(* IEC 61131-3 sources: Elmo_Master/Lasal_PRG/MotionTCPDemo/Class/TCPRT_DataManager, 1 file *)

(* ---- TCPRT_DataManager.st ---- *)
(*!
<Class
	Name               = "TCPRT_DataManager"
	Revision           = "0.0"
	RealtimeTask       = "true"
	CyclicTask         = "true"
	BackgroundTask     = "false"
	Sigmatek           = "false"
	OSInterface        = "false"
	HighPriority       = "false"
	Automatic          = "false"
	UpdateMode         = "Prescan"
	SharedCommandTable = "true"
	Objectsize         = "(678,0)">
	<Channels>
	</Channels>
	<Network Name="TCPRT_DataManager">
		<!-- List of Components in this network -->
		<Components>
			<Object
				Name       = "_base"
				Class      = "_SigTCPDataManager"
				Position   = "(218,120)"
				Visualized = "true"
				Remotely   = "true">
				<Channels>
					<Server Name="AcceptOfflineJobs" Value="1"/>
					<Server Name="ClassSvr"/>
					<Server Name="ComPort" Value="500"/>
					<Server Name="DeactivateCom" Value="0"/>
					<Server Name="DeleteJobs"/>
					<Server Name="LogEnable" Value="0"/>
					<Server Name="NoEntries"/>
					<Server Name="Online"/>
					<Server Name="ResetLogBuffer"/>
					<Server Name="TCPComm"/>
					<Client Name="ErrRuntime"/>
					<Client Name="InternConnection"/>
					<Client Name="IPtoConnect"/>
					<Client Name="LogFilter" Value="0"/>
					<Client Name="SizeOfComBufferRecv" Value="100 kB"/>
					<Client Name="SizeOfComBuffers" Value="100 kB"/>
					<Client Name="StationToConnect"/>
				</Channels>
			</Object>
		</Components>
		<Comments>
		</Comments>
		<!-- List of Connections in this network -->
		<Connections>
			<Connection Source="this.ClassSvr" Destination="_base.ClassSvr" Vertices="(1084,210),(912,210),"/>
			<Connection Source="this.NoEntries" Destination="_base.NoEntries" Vertices="(1084,270),(912,270),"/>
			<Connection Source="this.DeleteJobs" Destination="_base.DeleteJobs" Vertices="(1084,330),(912,330),"/>
			<Connection Source="this.AcceptOfflineJobs" Destination="_base.AcceptOfflineJobs" Vertices="(1084,390),(912,390),"/>
			<Connection Source="this.TCPComm" Destination="_base.TCPComm" Vertices="(1084,450),(912,510),"/>
			<Connection Source="this.ComPort" Destination="_base.ComPort" Vertices="(1084,510),(912,570),"/>
			<Connection Source="this.Online" Destination="_base.Online" Vertices="(1084,570),(912,630),"/>
			<Connection Source="this.LogEnable" Destination="_base.LogEnable" Vertices="(1084,630),(912,690),"/>
			<Connection Source="this.ResetLogBuffer" Destination="_base.ResetLogBuffer" Vertices="(1084,690),(912,750),"/>
			<Connection Source="this.DeactivateCom" Destination="_base.DeactivateCom" Vertices="(1084,750),(912,810),"/>
			<Connection Source="_base.InternConnection" Destination="this.InternConnection" Vertices="(218,210),(38,210),"/>
			<Connection Source="_base.IPtoConnect" Destination="this.IPtoConnect" Vertices="(218,270),(38,270),"/>
			<Connection Source="_base.StationToConnect" Destination="this.StationToConnect" Vertices="(218,330),(38,330),"/>
			<Connection Source="_base.LogFilter" Destination="this.LogFilter" Vertices="(218,390),(38,390),"/>
			<Connection Source="_base.ErrRuntime" Destination="this.ErrRuntime" Vertices="(218,450),(38,450),"/>
			<Connection Source="_base.SizeOfComBuffers" Destination="this.SizeOfComBuffers" Vertices="(218,510),(38,510),"/>
			<Connection Source="_base.SizeOfComBufferRecv" Destination="this.SizeOfComBufferRecv" Vertices="(218,570),(38,570),"/>
		</Connections>
		<!-- Headerfiles -->
		<Options>
		</Options>
	</Network>
</Class>
*)
#pragma using _SigTCPDataManager

TCPRT_DataManager : CLASS
: _SigTCPDataManager
  //Servers:
  //Clients:
  //Variables:
  //Functions:

	FUNCTION VIRTUAL GLOBAL RtWork
		VAR_INPUT
			EAX 	: UDINT;
		END_VAR
		VAR_OUTPUT
			state (EAX) 	: UDINT;
		END_VAR;
  //Tables:
	FUNCTION @STD
		VAR_OUTPUT
			ret_code	: CONFSTATES;
		END_VAR;
	FUNCTION GLOBAL TAB @CT_;
END_CLASS;

FUNCTION VIRTUAL GLOBAL TCPRT_DataManager::RtWork
	VAR_INPUT
		EAX 	: UDINT;
	END_VAR
	VAR_OUTPUT
		state (EAX) 	: UDINT;
	END_VAR

  state := _SigTCPDataManager::CyWork(EAX:=Eax);

END_FUNCTION
